// TwinCAT 3 PLC project Sample01
// ProgramVersion: 3.1.4022.3
// libraries:
//   Tc2_Standard, * (Beckhoff Automation GmbH)
//   Tc2_System, * (Beckhoff Automation GmbH)
//   Tc2_Utilities, * (Beckhoff Automation GmbH)
//   Tc3_Module, * (Beckhoff Automation GmbH)
// project tree:
//   / PlcTask.TcTTO
//   POUs/ F_AddMulti.TcPOU, F_AddAny.TcPOU, MAIN.TcPOU
// real-time tasks:
//   TASK PlcTask: cycle T#10ms, priority 20, ADS port 350

CONFIGURATION Sample01
    RESOURCE PLC ON TwinCAT3
        TASK PlcTask(INTERVAL := T#10ms, PRIORITY := 20);
        PROGRAM MAIN WITH PlcTask : MAIN;
    END_RESOURCE
END_CONFIGURATION

// ---- POUs/MAIN.TcPOU
PROGRAM MAIN
VAR
	sum			: LREAL;
	args		: ARRAY [1..4] OF T_Arg;
	a			: INT := 4567;
	b			: REAL := 3.1415;
	c			: DINT := 7032345;
	d			: USINT := 13;
END_VAR

args[1] := F_INT(a);
args[2] := F_REAL(b);
args[3] := F_DINT(c);
args[4] := F_USINT(d);
sum := F_AddMulti(args);

sum := F_AddAny(a, b) + F_AddAny(c, d);

END_PROGRAM

// ---- POUs/F_AddMulti.TcPOU
FUNCTION F_AddMulti : LREAL
VAR_IN_OUT
	aArgs		:	ARRAY [*] OF T_Arg;
END_VAR
VAR
	nIndex		:	DINT;
	aUSINT		:	USINT;
	aUINT		:	UINT;
	aINT		:	INT;
	aDINT		:	DINT;
	aREAL		:	REAL;
	aLREAL		:	LREAL;
END_VAR

F_AddMulti := 0.0;
FOR nIndex := LOWER_BOUND(aArgs, 1) TO UPPER_BOUND(aArgs, 1) DO
	CASE (aArgs[nIndex].eType) OF
		E_ArgType.ARGTYPE_USINT:
			MEMCPY(ADR(aUSINT), aArgs[nIndex].pData, aArgs[nIndex].cbLen);
			F_AddMulti := F_AddMulti + aUSINT;
		E_ArgType.ARGTYPE_UINT:
			MEMCPY(ADR(aUINT), aArgs[nIndex].pData, aArgs[nIndex].cbLen);
			F_AddMulti := F_AddMulti + aUINT;
		E_ArgType.ARGTYPE_INT:
			MEMCPY(ADR(aINT), aArgs[nIndex].pData, aArgs[nIndex].cbLen);
			F_AddMulti := F_AddMulti + aINT;
		E_ArgType.ARGTYPE_DINT:
			MEMCPY(ADR(aDINT), aArgs[nIndex].pData, aArgs[nIndex].cbLen);
			F_AddMulti := F_AddMulti + aDINT;
		E_ArgType.ARGTYPE_REAL:
			MEMCPY(ADR(aREAL), aArgs[nIndex].pData, aArgs[nIndex].cbLen);
			F_AddMulti := F_AddMulti + aREAL;
		E_ArgType.ARGTYPE_LREAL:
			MEMCPY(ADR(aLREAL), aArgs[nIndex].pData, aArgs[nIndex].cbLen);
			F_AddMulti := F_AddMulti + aLREAL;
	END_CASE
END_FOR

END_FUNCTION

// ---- POUs/F_AddAny.TcPOU
FUNCTION F_AddAny : LREAL
VAR_INPUT
	a			:	ANY;
	b			:	ANY;
END_VAR
VAR
	aUSINT		:	USINT;
	aUINT		:	UINT;
	aINT		:	INT;
	aDINT		:	DINT;
	aREAL		:	REAL;
	aLREAL		:	LREAL;

	bUSINT		:	USINT;
	bUINT		:	UINT;
	bINT		:	INT;
	bDINT		:	DINT;
	bREAL		:	REAL;
	bLREAL		:	LREAL;
END_VAR

CASE (a.TypeClass) OF
	__SYSTEM.TYPE_CLASS.TYPE_USINT:
		MEMCPY(ADR(aUSINT), a.pValue, TO_UDINT(a.diSize));
		F_AddAny := aUSINT;
	__SYSTEM.TYPE_CLASS.TYPE_UINT:
		MEMCPY(ADR(aUINT), a.pValue, TO_UDINT(a.diSize));
		F_AddAny := aUINT;
	__SYSTEM.TYPE_CLASS.TYPE_INT:
		MEMCPY(ADR(aINT), a.pValue, TO_UDINT(a.diSize));
		F_AddAny := aINT;
	__SYSTEM.TYPE_CLASS.TYPE_DINT:
		MEMCPY(ADR(aDINT), a.pValue, TO_UDINT(a.diSize));
		F_AddAny := aDINT;
	__SYSTEM.TYPE_CLASS.TYPE_REAL:
		MEMCPY(ADR(aREAL), a.pValue, TO_UDINT(a.diSize));
		F_AddAny := aREAL;
	__SYSTEM.TYPE_CLASS.TYPE_LREAL:
		MEMCPY(ADR(aLREAL), a.pValue, TO_UDINT(a.diSize));
		F_AddAny := aLREAL;
END_CASE

CASE (b.TypeClass) OF
	__SYSTEM.TYPE_CLASS.TYPE_USINT:
		MEMCPY(ADR(bUSINT), b.pValue, TO_UDINT(b.diSize));
		F_AddAny := F_AddAny + bUSINT;
	__SYSTEM.TYPE_CLASS.TYPE_UINT:
		MEMCPY(ADR(bUINT), b.pValue, TO_UDINT(b.diSize));
		F_AddAny := F_AddAny + bUINT;
	__SYSTEM.TYPE_CLASS.TYPE_INT:
		MEMCPY(ADR(bINT), b.pValue, TO_UDINT(b.diSize));
		F_AddAny := F_AddAny + bINT;
	__SYSTEM.TYPE_CLASS.TYPE_DINT:
		MEMCPY(ADR(bDINT), b.pValue, TO_UDINT(b.diSize));
		F_AddAny := F_AddAny + bDINT;
	__SYSTEM.TYPE_CLASS.TYPE_REAL:
		MEMCPY(ADR(bREAL), b.pValue, TO_UDINT(b.diSize));
		F_AddAny := F_AddAny + bREAL;
	__SYSTEM.TYPE_CLASS.TYPE_LREAL:
		MEMCPY(ADR(bLREAL), b.pValue, TO_UDINT(b.diSize));
		F_AddAny := F_AddAny + bLREAL;
END_CASE

END_FUNCTION
